FUNCTION_BLOCK xPlanarControl
VAR
	
	_PlanarMover			: ARRAY [1..MoverCount] OF MC_PlanarMover;
	_PlanarFeedback			: ARRAY [1..MoverCount] OF MC_PlanarFeedback;
	_MoveParameters			: ARRAY [1..MoverCount] OF ST_MoverParameters;
	
	_i						: BYTE;
	_LocalState				: BYTE;
	_InternalCounter		: UINT;
	_ErrorCount				: UINT;
	_CommandDone			: BOOL;
	
	_Enabled				: ARRAY [1.._MoverCount] OF BOOL;
	_Error					: ARRAY [1.._MoverCount] OF BOOL;
	_Busy					: ARRAY [1.._MoverCount] OF BOOL;
	_Done					: ARRAY [1.._MoverCount] OF BOOL;
	
	_Velocity				: LREAL := 2000;
	_Acceleration			: LREAL := 20000;
	_Deceleration			: LREAL := 20000;
	_Jerk					: LREAL := 200000;
	_NumberOfRotations		: UDINT := 5;
	
END_VAR
VAR CONSTANT
	
	_MoverCount				: BYTE := 2;

END_VAR

// NETWORK 1

METHOD CyclicUpdate : BOOL
VAR_INPUT
END_VAR

FOR _i := 1 TO _MoverCount DO
	
	_PlanarMover[_i].Update();
	_PlanarFeedback[_i].Update();
	
	IF _PlanarMover[_i].MCTOPLC.STD.State = 3 THEN
		_Enabled[_i] := TRUE;
	ELSE
		_Enabled[_i] := FALSE;
	END_IF

	_Error[_i] := _PlanarFeedback[_i].Error;
	_Busy[_i] := _PlanarFeedback[_i].Busy;
	_Done[_i] := _PlanarFeedback[_i].Done;
	
END_FOR

_MoveParameters[1].Options.useOrientation := TRUE;
_MoveParameters[1].Constraints.SetValuesVADJ(V := _Velocity, A := _Acceleration, D := _Deceleration, J := _Jerk);
_MoveParameters[1].rotateOptions.additionalTurns := _NumberOfRotations;
_MoveParameters[1].rotateOptions.direction := 1;

_MoveParameters[2].Options.useOrientation := TRUE;
_MoveParameters[2].Constraints.SetValuesVADJ(V := _Velocity, A := _Acceleration, D := _Deceleration, J := _Jerk);
_MoveParameters[2].rotateOptions.additionalTurns := _NumberOfRotations;
_MoveParameters[2].rotateOptions.direction := 3;
END_METHOD

METHOD PUBLIC DecreaseMoverHeight : BOOL
VAR_INPUT
END_VAR

// Movers go a bit low
	
CASE _LocalState OF
	
	0:
		_LocalState := 1;
	
	1:
		FOR _i := 1 TO _MoverCount DO
			_PlanarMover[_i].MoveZ
			(	
				commandFeedback		:= _PlanarFeedback[_i],
				targetPosition		:= 2.0,
				constraint			:= _MoveParameters[_i].Constraints
			);
		END_FOR
		_LocalState := 2;
	
	2:
		_CommandDone := TRUE;
		FOR _i := 1 TO _MoverCount DO
			IF NOT(_PlanarFeedback[_i].Done) THEN
				_CommandDone := FALSE;
				_InternalCounter := _InternalCounter + 1;
			END_IF
		END_FOR
		
		IF _InternalCounter >= 10000 THEN
			_LocalState := 0;
			_InternalCounter := 0;
			DecreaseMoverHeight := FALSE;
		END_IF
		
		IF _CommandDone THEN
			_CommandDone := FALSE;
			_InternalCounter := 0;
			_LocalState := 2;
		END_IF

	3:
		DecreaseMoverHeight := TRUE;
		_LocalState := 0;

END_CASE
END_METHOD

METHOD DetectErrors : BOOL
VAR_INPUT
END_VAR

FOR _i := 1 TO _MoverCount DO
	IF _PlanarMover[_i].Error THEN
		_Error[_i] := TRUE;
		_ErrorCount := _ErrorCount + 1;
		DetectErrors := TRUE;
	END_IF
END_FOR
END_METHOD

METHOD DisableMovers : BOOL
VAR_INPUT
END_VAR

CASE _LocalState OF
	
	0:
		FOR _i := 1 TO _MoverCount DO
			_PlanarMover[_i].Disable(_PlanarFeedback[_i]);
		END_FOR
		_LocalState := 1;
	
	1:
		_CommandDone := TRUE;
		FOR _i := 1 TO _MoverCount DO
			IF NOT(_PlanarFeedback[_i].Done) THEN
				_CommandDone := FALSE;
				_InternalCounter := _InternalCounter + 1;
			END_IF
		END_FOR
		
		IF _InternalCounter >= 10000 THEN
			_LocalState := 0;
			_InternalCounter := 0;
			DisableMovers := FALSE;
		END_IF
		
		IF _CommandDone THEN
			_CommandDone := FALSE;
			_InternalCounter := 0;
			_LocalState := 2;
		END_IF
	
	2:
		_LocalState := 0;
		DisableMovers := TRUE;

END_CASE
END_METHOD

METHOD EnableMovers : BOOL
VAR_INPUT
END_VAR

CASE _LocalState OF
	
	0:
		FOR _i := 1 TO _MoverCount DO
			_PlanarMover[_i].Enable(_PlanarFeedback[_i]);
		END_FOR
		_LocalState := 1;
	
	1:
		_CommandDone := TRUE;
		FOR _i := 1 TO _MoverCount DO
			IF NOT(_PlanarFeedback[_i].Done) THEN
				_CommandDone := FALSE;
				_InternalCounter := _InternalCounter + 1;
			END_IF
		END_FOR
		
		IF _InternalCounter >= 10000 THEN
			_LocalState := 0;
			_InternalCounter := 0;
			EnableMovers := FALSE;
		END_IF
		
		IF _CommandDone THEN
			_CommandDone := FALSE;
			_InternalCounter := 0;
			_LocalState := 2;
		END_IF
	
	2:
		_LocalState := 0;
		EnableMovers := TRUE;

END_CASE
END_METHOD

METHOD PUBLIC FollowTileEdge : BOOL
VAR_INPUT
END_VAR

// Movers move to edge of tiles and follow the perimeter, then move to home
	
	CASE _LocalState OF
		
		0:
			_LocalState := 1;
	
		1:
			_MoveParameters[1].targetPosition.x := 180;
			_MoveParameters[1].targetPosition.y := 183;
			_MoveParameters[2].targetPosition.x := 296;
			_MoveParameters[2].targetPosition.y := 183;
			_LocalState := 2;
		
		2:
			FOR _i := 1 TO _MoverCount DO
				_PlanarMover[_i].MoveToPosition
				(
					commandFeedback 	:= _PlanarFeedback[_i],
					targetPosition 		:= _MoveParameters[_i].targetPosition,
					constraint 			:= _MoveParameters[_i].Constraints,
					options 			:= _MoveParameters[_i].Options
				);
			END_FOR
			_LocalState := 3;
		
		3:
			_CommandDone := TRUE;
			FOR _i := 1 TO _MoverCount DO
				IF NOT(_PlanarFeedback[_i].Done) THEN
					_CommandDone := FALSE;
					_InternalCounter := _InternalCounter + 1;
				END_IF
			END_FOR
			
			IF _InternalCounter >= 10000 THEN
				_LocalState := 0;
				_InternalCounter := 0;
				FollowTileEdge := FALSE;
			END_IF
			
			IF _CommandDone THEN
				_CommandDone := FALSE;
				_InternalCounter := 0;
				_LocalState := 4;
			END_IF
	
		4:
			_MoveParameters[1].targetPosition.x := 57;
			_MoveParameters[1].targetPosition.y := 183;
			_MoveParameters[2].targetPosition.x := 423;
			_MoveParameters[2].targetPosition.y := 183;
			_LocalState := 5;
		
		5:
			FOR _i := 1 TO _MoverCount DO
				_PlanarMover[_i].MoveToPosition
				(
					commandFeedback 	:= _PlanarFeedback[_i],
					targetPosition 		:= _MoveParameters[_i].targetPosition,
					constraint 			:= _MoveParameters[_i].Constraints,
					options 			:= _MoveParameters[_i].Options
				);
			END_FOR
			_LocalState := 6;
		
		6:
			_CommandDone := TRUE;
			FOR _i := 1 TO _MoverCount DO
				IF NOT(_PlanarFeedback[_i].Done) THEN
					_CommandDone := FALSE;
					_InternalCounter := _InternalCounter + 1;
				END_IF
			END_FOR
			
			IF _InternalCounter >= 10000 THEN
				_LocalState := 0;
				_InternalCounter := 0;
				FollowTileEdge := FALSE;
			END_IF
			
			IF _CommandDone THEN
				_CommandDone := FALSE;
				_InternalCounter := 0;
				_LocalState := 7;
			END_IF
			
		7:
			_MoveParameters[1].targetPosition.x := 57;
			_MoveParameters[1].targetPosition.y := 57;
			_MoveParameters[2].targetPosition.x := 423;
			_MoveParameters[2].targetPosition.y := 57;
			_LocalState := 8;
		
		8:
			FOR _i := 1 TO _MoverCount DO
				_PlanarMover[_i].MoveToPosition
				(
					commandFeedback 	:= _PlanarFeedback[_i],
					targetPosition 		:= _MoveParameters[_i].targetPosition,
					constraint 			:= _MoveParameters[_i].Constraints,
					options 			:= _MoveParameters[_i].Options
				);
			END_FOR
			_LocalState := 9;
		
		9:
			_CommandDone := TRUE;
			FOR _i := 1 TO _MoverCount DO
				IF NOT(_PlanarFeedback[_i].Done) THEN
					_CommandDone := FALSE;
					_InternalCounter := _InternalCounter + 1;
				END_IF
			END_FOR
			
			IF _InternalCounter >= 10000 THEN
				_LocalState := 0;
				_InternalCounter := 0;
				FollowTileEdge := FALSE;
			END_IF
			
			IF _CommandDone THEN
				_CommandDone := FALSE;
				_InternalCounter := 0;
				_LocalState := 10;
			END_IF
			
		10:
			_MoveParameters[1].targetPosition.x := 180;
			_MoveParameters[1].targetPosition.y := 57;
			_MoveParameters[2].targetPosition.x := 296;
			_MoveParameters[2].targetPosition.y := 57;
			_LocalState := 11;
		
		11:
			FOR _i := 1 TO _MoverCount DO
				_PlanarMover[_i].MoveToPosition
				(
					commandFeedback 	:= _PlanarFeedback[_i],
					targetPosition 		:= _MoveParameters[_i].targetPosition,
					constraint 			:= _MoveParameters[_i].Constraints,
					options 			:= _MoveParameters[_i].Options
				);
			END_FOR
			_LocalState := 12;
		
		12:
			_CommandDone := TRUE;
			FOR _i := 1 TO _MoverCount DO
				IF NOT(_PlanarFeedback[_i].Done) THEN
					_CommandDone := FALSE;
					_InternalCounter := _InternalCounter + 1;
				END_IF
			END_FOR
			
			IF _InternalCounter >= 10000 THEN
				_LocalState := 0;
				_InternalCounter := 0;
				FollowTileEdge := FALSE;
			END_IF
			
			IF _CommandDone THEN
				_CommandDone := FALSE;
				_InternalCounter := 0;
				_LocalState := 13;
			END_IF
			
		13:
			_MoveParameters[1].targetPosition.x := 120;
			_MoveParameters[1].targetPosition.y := 120;
			_MoveParameters[2].targetPosition.x := 360;
			_MoveParameters[2].targetPosition.y := 120;
			_LocalState := 14;
		
		14:
			FOR _i := 1 TO _MoverCount DO
				_PlanarMover[_i].MoveToPosition
				(
					commandFeedback 	:= _PlanarFeedback[_i],
					targetPosition 		:= _MoveParameters[_i].targetPosition,
					constraint 			:= _MoveParameters[_i].Constraints,
					options 			:= _MoveParameters[_i].Options
				);
			END_FOR
			_LocalState := 15;
		
		15:
			_CommandDone := TRUE;
			FOR _i := 1 TO _MoverCount DO
				IF NOT(_PlanarFeedback[_i].Done) THEN
					_CommandDone := FALSE;
					_InternalCounter := _InternalCounter + 1;
				END_IF
			END_FOR
			
			IF _InternalCounter >= 10000 THEN
				_LocalState := 0;
				_InternalCounter := 0;
				FollowTileEdge := FALSE;
			END_IF
			
			IF _CommandDone THEN
				_CommandDone := FALSE;
				_InternalCounter := 0;
				_LocalState := 16;
			END_IF
			
		16:
			FollowTileEdge := TRUE;
			_LocalState := 0;
			
	END_CASE
END_METHOD

METHOD PUBLIC Home : BOOL
VAR_INPUT
END_VAR

// Move movers to the middle of tiles.
	
CASE _LocalState OF
		
	0:
		_LocalState := 1;
		
	1:
		_MoveParameters[1].targetPosition.x := 120;
		_MoveParameters[1].targetPosition.y := 120;
		_MoveParameters[2].targetPosition.x := 360;
		_MoveParameters[2].targetPosition.y := 120;
		_LocalState := 2;
		
	2:
		FOR _i := 1 TO _MoverCount DO
			_PlanarMover[_i].MoveToPosition
			(
				commandFeedback 	:= _PlanarFeedback[_i],
				targetPosition 		:= _MoveParameters[_i].targetPosition,
				constraint 			:= _MoveParameters[_i].Constraints,
				options 			:= _MoveParameters[_i].Options
			);
		END_FOR
		_LocalState := 3;
		
	3:
		_CommandDone := TRUE;
		FOR _i := 1 TO _MoverCount DO
			IF NOT(_PlanarFeedback[_i].Done) THEN
				_CommandDone := FALSE;
				_InternalCounter := _InternalCounter + 1;
			END_IF
		END_FOR
		
		IF _InternalCounter >= 10000 THEN
			_LocalState := 0;
			_InternalCounter := 0;
			Home := FALSE;
		END_IF
		
		IF _CommandDone THEN
			_CommandDone := FALSE;
			_InternalCounter := 0;
			_LocalState := 4;
		END_IF
		
	4:
		Home := TRUE;
		_LocalState := 0;
		
		
END_CASE
END_METHOD

PROPERTY MoverAcceleration : LREAL
GET
MoverAcceleration := _Acceleration;
END_GET
SET
IF (MoverAcceleration <= 0) OR (MoverAcceleration > 20000) THEN
	_Acceleration := 20000;
ELSE
	_Acceleration := MoverAcceleration;
END_IF
END_SET
END_PROPERTY

PROPERTY MoverDeceleration : LREAL
GET
MoverDeceleration := _Deceleration;
END_GET
SET
IF (MoverDeceleration <= 0) OR (MoverDeceleration > 20000) THEN
	_Deceleration := 20000;
ELSE
	_Deceleration := MoverDeceleration;
END_IF
END_SET
END_PROPERTY

PROPERTY MoverJerk : LREAL
GET
MoverJerk := _Jerk;
END_GET
SET
IF (MoverJerk <= 0) OR (MoverJerk > 200000) THEN
	_Jerk := 200000;
ELSE
	_Jerk := MoverJerk;
END_IF
END_SET
END_PROPERTY

PROPERTY MoverVelocity : LREAL
GET
MoverVelocity := _Velocity;
END_GET
SET
IF (MoverVelocity <= 0) OR (MoverVelocity > 2000) THEN
	_Velocity := 2000;
ELSE
	_Velocity := MoverVelocity;
END_IF
END_SET
END_PROPERTY

PROPERTY NumberOfRotations : UDINT
GET
NumberOfRotations := _NumberOfRotations;
END_GET
SET
IF (NumberOfRotations <= 0) THEN
	_NumberOfRotations := 1;
ELSE
	_NumberOfRotations := NumberOfRotations;
END_IF
END_SET
END_PROPERTY

METHOD ResetErrors : BOOL
VAR_INPUT
END_VAR

CASE _LocalState OF
	
	0: 
		FOR _i := 1 TO _MoverCount DO
			_PlanarMover[_i].Reset(_PlanarFeedback[_i]);
		END_FOR
		_LocalState := 1;
	
	1:	
		_CommandDone := TRUE;
		FOR _i := 1 TO _MoverCount DO
			IF NOT(_PlanarFeedback[_i].Done) THEN
				_CommandDone := FALSE;
				_InternalCounter := _InternalCounter + 1;
			END_IF
		END_FOR
		
		IF _InternalCounter >= 10000 THEN
			_LocalState := 0;
			_InternalCounter := 0;
			ResetErrors := FALSE;
		END_IF
		
		IF _CommandDone THEN
			_CommandDone := FALSE;
			_InternalCounter := 0;
			_LocalState := 2;
		END_IF

			
	2:
		_LocalState := 0;
		ResetErrors := TRUE;
	
END_CASE
END_METHOD

METHOD PUBLIC Spin : BOOL
VAR_INPUT
END_VAR

// Movers spin

CASE _LocalState OF
	
	0:
		_LocalState := 1;

	
	1:
		FOR _i := 1 TO _MoverCount DO
			_PlanarMover[_i].MoveC
			(	
				commandFeedback		:= _PlanarFeedback[_i],
				targetPosition		:= 0,
				constraint			:= _MoveParameters[_i].Constraints,
				options 			:= _MoveParameters[_i].rotateOptions
			);
		END_FOR
		_LocalState := 2;
	
	2:
		_CommandDone := TRUE;
		FOR _i := 1 TO _MoverCount DO
			IF NOT(_PlanarFeedback[_i].Done) THEN
				_CommandDone := FALSE;
				_InternalCounter := _InternalCounter + 1;
			END_IF
		END_FOR
		
		IF _InternalCounter >= 10000 THEN
			_LocalState := 0;
			_InternalCounter := 0;
			Spin := FALSE;
		END_IF
		
		IF _CommandDone THEN
			_CommandDone := FALSE;
			_InternalCounter := 0;
			_LocalState := 2;
		END_IF
		
	3:
		Spin := TRUE;
		_LocalState := 0;
	
END_CASE
END_METHOD

METHOD PUBLIC SwapPlaces : BOOL
VAR_INPUT
END_VAR

// Movers swap tiles, then swap back, then move to home
	
CASE _LocalState OF
	
	0:
		_LocalState := 1;

	1:
		_MoveParameters[1].targetPosition.x := 175;
		_MoveParameters[1].targetPosition.y := 183;
		_MoveParameters[2].targetPosition.x := 301;
		_MoveParameters[2].targetPosition.y := 57;
		_LocalState := 2;
	
	2:
		FOR _i := 1 TO _MoverCount DO
			_PlanarMover[_i].MoveToPosition
			(
				commandFeedback 	:= _PlanarFeedback[_i],
				targetPosition 		:= _MoveParameters[_i].targetPosition,
				constraint 			:= _MoveParameters[_i].Constraints,
				options 			:= _MoveParameters[_i].Options
			);
		END_FOR
		_LocalState := 3;
	
	3:
		_CommandDone := TRUE;
		FOR _i := 1 TO _MoverCount DO
			IF NOT(_PlanarFeedback[_i].Done) THEN
				_CommandDone := FALSE;
				_InternalCounter := _InternalCounter + 1;
			END_IF
		END_FOR
		
		IF _InternalCounter >= 10000 THEN
			_LocalState := 0;
			_InternalCounter := 0;
			SwapPlaces := FALSE;
		END_IF
		
		IF _CommandDone THEN
			_CommandDone := FALSE;
			_InternalCounter := 0;
			_LocalState := 4;
		END_IF

	4:
		_MoveParameters[1].targetPosition.x := 301;
		_MoveParameters[1].targetPosition.y := 183;
		_MoveParameters[2].targetPosition.x := 175;
		_MoveParameters[2].targetPosition.y := 57;
		_LocalState := 5;
	
	5:
		FOR _i := 1 TO _MoverCount DO
			_PlanarMover[_i].MoveToPosition
			(
				commandFeedback 	:= _PlanarFeedback[_i],
				targetPosition 		:= _MoveParameters[_i].targetPosition,
				constraint 			:= _MoveParameters[_i].Constraints,
				options 			:= _MoveParameters[_i].Options
			);
		END_FOR
		_LocalState := 6;
	
	6:
		_CommandDone := TRUE;
		FOR _i := 1 TO _MoverCount DO
			IF NOT(_PlanarFeedback[_i].Done) THEN
				_CommandDone := FALSE;
				_InternalCounter := _InternalCounter + 1;
			END_IF
		END_FOR
		
		IF _InternalCounter >= 10000 THEN
			_LocalState := 0;
			_InternalCounter := 0;
			SwapPlaces := FALSE;
		END_IF
		
		IF _CommandDone THEN
			_CommandDone := FALSE;
			_InternalCounter := 0;
			_LocalState := 7;
		END_IF
		
	7:
		_MoveParameters[1].targetPosition.x := 301;
		_MoveParameters[1].targetPosition.y := 57;
		_MoveParameters[2].targetPosition.x := 175;
		_MoveParameters[2].targetPosition.y := 183;
		_LocalState := 8;
	
	8:
		FOR _i := 1 TO _MoverCount DO
			_PlanarMover[_i].MoveToPosition
			(
				commandFeedback 	:= _PlanarFeedback[_i],
				targetPosition 		:= _MoveParameters[_i].targetPosition,
				constraint 			:= _MoveParameters[_i].Constraints,
				options 			:= _MoveParameters[_i].Options
			);
		END_FOR
		_LocalState := 9;
	
	9:
		_CommandDone := TRUE;
		FOR _i := 1 TO _MoverCount DO
			IF NOT(_PlanarFeedback[_i].Done) THEN
				_CommandDone := FALSE;
				_InternalCounter := _InternalCounter + 1;
			END_IF
		END_FOR
		
		IF _InternalCounter >= 10000 THEN
			_LocalState := 0;
			_InternalCounter := 0;
			SwapPlaces := FALSE;
		END_IF
		
		IF _CommandDone THEN
			_CommandDone := FALSE;
			_InternalCounter := 0;
			_LocalState := 10;
		END_IF
		
	10:
		_MoveParameters[1].targetPosition.x := 175;
		_MoveParameters[1].targetPosition.y := 57;
		_MoveParameters[2].targetPosition.x := 301;
		_MoveParameters[2].targetPosition.y := 183;
		_LocalState := 11;
	
	11:
		FOR _i := 1 TO _MoverCount DO
			_PlanarMover[_i].MoveToPosition
			(
				commandFeedback 	:= _PlanarFeedback[_i],
				targetPosition 		:= _MoveParameters[_i].targetPosition,
				constraint 			:= _MoveParameters[_i].Constraints,
				options 			:= _MoveParameters[_i].Options
			);
		END_FOR
		_LocalState := 12;
	
	12:
		_CommandDone := TRUE;
		FOR _i := 1 TO _MoverCount DO
			IF NOT(_PlanarFeedback[_i].Done) THEN
				_CommandDone := FALSE;
				_InternalCounter := _InternalCounter + 1;
			END_IF
		END_FOR
		
		IF _InternalCounter >= 10000 THEN
			_LocalState := 0;
			_InternalCounter := 0;
			SwapPlaces := FALSE;
		END_IF
		
		IF _CommandDone THEN
			_CommandDone := FALSE;
			_InternalCounter := 0;
			_LocalState := 13;
		END_IF
		
	13:
		_MoveParameters[1].targetPosition.x := 120;
		_MoveParameters[1].targetPosition.y := 120;
		_MoveParameters[2].targetPosition.x := 360;
		_MoveParameters[2].targetPosition.y := 120;
		_LocalState := 14;
	
	14:
		FOR _i := 1 TO _MoverCount DO
			_PlanarMover[_i].MoveToPosition
			(
				commandFeedback 	:= _PlanarFeedback[_i],
				targetPosition 		:= _MoveParameters[_i].targetPosition,
				constraint 			:= _MoveParameters[_i].Constraints,
				options 			:= _MoveParameters[_i].Options
			);
		END_FOR
		_LocalState := 15;
	
	15:
		_CommandDone := TRUE;
		FOR _i := 1 TO _MoverCount DO
			IF NOT(_PlanarFeedback[_i].Done) THEN
				_CommandDone := FALSE;
				_InternalCounter := _InternalCounter + 1;
			END_IF
		END_FOR
		
		IF _InternalCounter >= 10000 THEN
			_LocalState := 0;
			_InternalCounter := 0;
			SwapPlaces := FALSE;
		END_IF
		
		IF _CommandDone THEN
			_CommandDone := FALSE;
			_InternalCounter := 0;
			_LocalState := 16;
		END_IF
		
	16:
		SwapPlaces := TRUE;
		_LocalState := 0;
		
END_CASE
END_METHOD

METHOD PUBLIC Tilt : BOOL
VAR_INPUT
END_VAR

// Movers tilt

CASE _LocalState OF
	
	0:
		_LocalState := 1;
		
	1:
		FOR _i := 1 TO _MoverCount DO
			_PlanarMover[_i].MoveZ
			(	
				commandFeedback		:= _PlanarFeedback[_i],
				targetPosition		:= 5.0,
				constraint			:= _MoveParameters[_i].Constraints
			);
		END_FOR
		_LocalState := 2;
	
	2:
		_CommandDone := TRUE;
		FOR _i := 1 TO _MoverCount DO
			IF NOT(_PlanarFeedback[_i].Done) THEN
				_CommandDone := FALSE;
				_InternalCounter := _InternalCounter + 1;
			END_IF
		END_FOR
		
		IF _InternalCounter >= 10000 THEN
			_LocalState := 0;
			_InternalCounter := 0;
			Tilt := FALSE;
		END_IF
		
		IF _CommandDone THEN
			_CommandDone := FALSE;
			_InternalCounter := 0;
			_LocalState := 3;
		END_IF

	
	3:
		FOR _i := 1 TO xPlanarLink.MoverCount DO
			xPlanarLink.PlanarMover[_i].MoveA
			(	
				commandFeedback		:= xPlanarLink.PlanarFeedback[_i],
				targetPosition		:= 4.0,
				constraint			:= _MoveParameters[_i].Constraints
			);
		END_FOR
		_LocalState := 4;
	
	4:
		_CommandDone := TRUE;
		FOR _i := 1 TO _MoverCount DO
			IF NOT(_PlanarFeedback[_i].Done) THEN
				_CommandDone := FALSE;
				_InternalCounter := _InternalCounter + 1;
			END_IF
		END_FOR
		
		IF _InternalCounter >= 10000 THEN
			_LocalState := 0;
			_InternalCounter := 0;
			Tilt := FALSE;
		END_IF
		
		IF _CommandDone THEN
			_CommandDone := FALSE;
			_InternalCounter := 0;
			_LocalState := 5;
		END_IF
		
	5:
		FOR _i := 1 TO _MoverCount DO
			_PlanarMover[_i].MoveA
			(	
				commandFeedback		:= _PlanarFeedback[_i],
				targetPosition		:= -4.0,
				constraint			:= _MoveParameters[_i].Constraints
			);
		END_FOR
		_LocalState := 6;
	
	6:
		_CommandDone := TRUE;
		FOR _i := 1 TO _MoverCount DO
			IF NOT(_PlanarFeedback[_i].Done) THEN
				_CommandDone := FALSE;
				_InternalCounter := _InternalCounter + 1;
			END_IF
		END_FOR
		
		IF _InternalCounter >= 10000 THEN
			_LocalState := 0;
			_InternalCounter := 0;
			Tilt := FALSE;
		END_IF
		
		IF _CommandDone THEN
			_CommandDone := FALSE;
			_InternalCounter := 0;
			_LocalState := 7;
		END_IF
	
	7:
		FOR _i := 1 TO _MoverCount DO
			_PlanarMover[_i].MoveA
			(	
				commandFeedback		:= _PlanarFeedback[_i],
				targetPosition		:= 0.0,
				constraint			:= _MoveParameters[_i].Constraints
			);
		END_FOR
		_LocalState := 8;
	
	8:
		_CommandDone := TRUE;
		FOR _i := 1 TO _MoverCount DO
			IF NOT(_PlanarFeedback[_i].Done) THEN
				_CommandDone := FALSE;
				_InternalCounter := _InternalCounter + 1;
			END_IF
		END_FOR
		
		IF _InternalCounter >= 10000 THEN
			_LocalState := 0;
			_InternalCounter := 0;
			Tilt := FALSE;
		END_IF
		
		IF _CommandDone THEN
			_CommandDone := FALSE;
			_InternalCounter := 0;
			_LocalState := 9;
		END_IF
		
	9:
		FOR _i := 1 TO _MoverCount DO
			_PlanarMover[_i].MoveB
			(	
				commandFeedback		:= _PlanarFeedback[_i],
				targetPosition		:= 4.0,
				constraint			:= _MoveParameters[_i].Constraints
			);
		END_FOR
		_LocalState := 10;
	
	10:
		_CommandDone := TRUE;
		FOR _i := 1 TO _MoverCount DO
			IF NOT(_PlanarFeedback[_i].Done) THEN
				_CommandDone := FALSE;
				_InternalCounter := _InternalCounter + 1;
			END_IF
		END_FOR
		
		IF _InternalCounter >= 10000 THEN
			_LocalState := 0;
			_InternalCounter := 0;
			Tilt := FALSE;
		END_IF
		
		IF _CommandDone THEN
			_CommandDone := FALSE;
			_InternalCounter := 0;
			_LocalState := 11;
		END_IF
		
	11:
		FOR _i := 1 TO _MoverCount DO
			_PlanarMover[_i].MoveB
			(	
				commandFeedback		:= _PlanarFeedback[_i],
				targetPosition		:= -4.0,
				constraint			:= _MoveParameters[_i].Constraints
			);
		END_FOR
		_LocalState := 12;
	
	12:
		_CommandDone := TRUE;
		FOR _i := 1 TO _MoverCount DO
			IF NOT(_PlanarFeedback[_i].Done) THEN
				_CommandDone := FALSE;
				_InternalCounter := _InternalCounter + 1;
			END_IF
		END_FOR
		
		IF _InternalCounter >= 10000 THEN
			_LocalState := 0;
			_InternalCounter := 0;
			Tilt := FALSE;
		END_IF
		
		IF _CommandDone THEN
			_CommandDone := FALSE;
			_InternalCounter := 0;
			_LocalState := 13;
		END_IF
	
	13:
		FOR _i := 1 TO _MoverCount DO
			_PlanarMover[_i].MoveB
			(	
				commandFeedback		:= _PlanarFeedback[_i],
				targetPosition		:= 0.0,
				constraint			:= _MoveParameters[_i].Constraints
			);
		END_FOR
		_LocalState := 14;
	
	14:
		_CommandDone := TRUE;
		FOR _i := 1 TO _MoverCount DO
			IF NOT(_PlanarFeedback[_i].Done) THEN
				_CommandDone := FALSE;
				_InternalCounter := _InternalCounter + 1;
			END_IF
		END_FOR
		
		IF _InternalCounter >= 10000 THEN
			_LocalState := 0;
			_InternalCounter := 0;
			Tilt := FALSE;
		END_IF
		
		IF _CommandDone THEN
			_CommandDone := FALSE;
			_InternalCounter := 0;
			_LocalState := 15;
		END_IF
		
	15:
		FOR _i := 1 TO _MoverCount DO
			_PlanarMover[_i].MoveZ
			(	
				commandFeedback		:= _PlanarFeedback[_i],
				targetPosition		:= 2.0,
				constraint			:= _MoveParameters[_i].Constraints
			);
		END_FOR
		_LocalState := 16;
	
	16:
		_CommandDone := TRUE;
		FOR _i := 1 TO _MoverCount DO
			IF NOT(_PlanarFeedback[_i].Done) THEN
				_CommandDone := FALSE;
				_InternalCounter := _InternalCounter + 1;
			END_IF
		END_FOR
		
		IF _InternalCounter >= 10000 THEN
			_LocalState := 0;
			_InternalCounter := 0;
			Tilt := FALSE;
		END_IF
		
		IF _CommandDone THEN
			_CommandDone := FALSE;
			_InternalCounter := 0;
			_LocalState := 17;
		END_IF
		
	17:
		Tilt := TRUE;
		_LocalState := 0;
	
END_CASE
END_METHOD

METHOD PUBLIC VaryMoverHeight : BOOL
VAR_INPUT
END_VAR

// Movers go a bit high

CASE _LocalState OF
	
	0:
		_LocalState := 1;
	
	1:
		FOR _i := 1 TO _MoverCount DO
			_PlanarMover[_i].MoveZ
			(	
				commandFeedback		:= _PlanarFeedback[_i],
				targetPosition		:= 5.0,
				constraint			:= _MoveParameters[_i].Constraints
			);
		END_FOR
		_LocalState := 2;
	
	2:
		_CommandDone := TRUE;
		FOR _i := 1 TO _MoverCount DO
			IF NOT(_PlanarFeedback[_i].Done) THEN
				_CommandDone := FALSE;
				_InternalCounter := _InternalCounter + 1;
			END_IF
		END_FOR
		
		IF _InternalCounter >= 10000 THEN
			_LocalState := 0;
			_InternalCounter := 0;
			VaryMoverHeight := FALSE;
		END_IF
		
		IF _CommandDone THEN
			_CommandDone := FALSE;
			_InternalCounter := 0;
			_LocalState := 3;
		END_IF
		
	3:
		FOR _i := 1 TO _MoverCount DO
			_PlanarMover[_i].MoveZ
			(	
				commandFeedback		:= _PlanarFeedback[_i],
				targetPosition		:= 2.0,
				constraint			:= _MoveParameters[_i].Constraints
			);
		END_FOR
		_LocalState := 4;
	
	4:
		_CommandDone := TRUE;
		FOR _i := 1 TO _MoverCount DO
			IF NOT(_PlanarFeedback[_i].Done) THEN
				_CommandDone := FALSE;
				_InternalCounter := _InternalCounter + 1;
			END_IF
		END_FOR
		
		IF _InternalCounter >= 10000 THEN
			_LocalState := 0;
			_InternalCounter := 0;
			VaryMoverHeight := FALSE;
		END_IF
		
		IF _CommandDone THEN
			_CommandDone := FALSE;
			_InternalCounter := 0;
			_LocalState := 5;
		END_IF
		
	5:
		FOR _i := 1 TO _MoverCount DO
			_PlanarMover[_i].MoveZ
			(	
				commandFeedback		:= _PlanarFeedback[_i],
				targetPosition		:= 5.0,
				constraint			:= _MoveParameters[_i].Constraints
			);
		END_FOR
		_LocalState := 6;
	
	6:
		_CommandDone := TRUE;
		FOR _i := 1 TO _MoverCount DO
			IF NOT(_PlanarFeedback[_i].Done) THEN
				_CommandDone := FALSE;
				_InternalCounter := _InternalCounter + 1;
			END_IF
		END_FOR
		
		IF _InternalCounter >= 10000 THEN
			_LocalState := 0;
			_InternalCounter := 0;
			VaryMoverHeight := FALSE;
		END_IF
		
		IF _CommandDone THEN
			_CommandDone := FALSE;
			_InternalCounter := 0;
			_LocalState := 7;
		END_IF
		
	7:
		FOR _i := 1 TO _MoverCount DO
			_PlanarMover[_i].MoveZ
			(	
				commandFeedback		:= _PlanarFeedback[_i],
				targetPosition		:= 2.0,
				constraint			:= _MoveParameters[_i].Constraints
			);
		END_FOR
		_LocalState := 8;
	
	8:
		_CommandDone := TRUE;
		FOR _i := 1 TO _MoverCount DO
			IF NOT(_PlanarFeedback[_i].Done) THEN
				_CommandDone := FALSE;
				_InternalCounter := _InternalCounter + 1;
			END_IF
		END_FOR
		
		IF _InternalCounter >= 10000 THEN
			_LocalState := 0;
			_InternalCounter := 0;
			VaryMoverHeight := FALSE;
		END_IF
		
		IF _CommandDone THEN
			_CommandDone := FALSE;
			_InternalCounter := 0;
			_LocalState := 9;
		END_IF
		
	9:
		FOR _i := 1 TO _MoverCount DO
			_PlanarMover[_i].MoveZ
			(	
				commandFeedback		:= _PlanarFeedback[_i],
				targetPosition		:= 5.0,
				constraint			:= _MoveParameters[_i].Constraints
			);
		END_FOR
		_LocalState := 10;
	
	10:
		_CommandDone := TRUE;
		FOR _i := 1 TO _MoverCount DO
			IF NOT(_PlanarFeedback[_i].Done) THEN
				_CommandDone := FALSE;
				_InternalCounter := _InternalCounter + 1;
			END_IF
		END_FOR
		
		IF _InternalCounter >= 10000 THEN
			_LocalState := 0;
			_InternalCounter := 0;
			VaryMoverHeight := FALSE;
		END_IF
		
		IF _CommandDone THEN
			_CommandDone := FALSE;
			_InternalCounter := 0;
			_LocalState := 11;
		END_IF

	11:
		FOR _i := 1 TO _MoverCount DO
			_PlanarMover[_i].MoveZ
			(	
				commandFeedback		:= _PlanarFeedback[_i],
				targetPosition		:= 2.0,
				constraint			:= _MoveParameters[_i].Constraints
			);
		END_FOR
		_LocalState := 12;
	
	12:
		_CommandDone := TRUE;
		FOR _i := 1 TO _MoverCount DO
			IF NOT(_PlanarFeedback[_i].Done) THEN
				_CommandDone := FALSE;
				_InternalCounter := _InternalCounter + 1;
			END_IF
		END_FOR
		
		IF _InternalCounter >= 10000 THEN
			_LocalState := 0;
			_InternalCounter := 0;
			VaryMoverHeight := FALSE;
		END_IF
		
		IF _CommandDone THEN
			_CommandDone := FALSE;
			_InternalCounter := 0;
			_LocalState := 13;
		END_IF
		
	13:
		VaryMoverHeight := TRUE;
		_LocalState := 0;

END_CASE
END_METHOD

END_FUNCTION_BLOCK

(* stored: Version 1.1.0.1, ProductVersion 3.1.4024.12
   POU xPlanarControl: Id {418f5a4e-4a80-43af-8346-cac2175cf5a1}, SpecialFunc None
   Folder Movements 2-Tile: Id {564f56f8-bb5c-4eca-8a56-c64a7594c15d}
   Folder Movements General: Id {aee95a18-140d-4ee9-ac40-69e7d69f9acf}
   Folder Power and Utility: Id {c5ba77ca-a5ce-43bc-a81f-9b9628e1d54c}
   Folder Properties: Id {0453768e-2223-4ce2-b57c-26f2fb086bed}
   Method CyclicUpdate: Id {c7e9e683-b8ab-4217-b047-2e15baa6471c}
   Method DecreaseMoverHeight: Id {d9c1f541-a92b-457b-b498-ae0f9078990c}
   Method DetectErrors: Id {daaeb43c-d127-4004-8d5e-5bf5a68f458b}
   Method DisableMovers: Id {425fd2bc-6f54-4fce-935d-1f0a1dc8c22b}
   Method EnableMovers: Id {ecc31ae1-6e60-4543-ab06-14adb5849eca}
   Method FollowTileEdge: Id {87cfbbfe-b39c-4b51-8245-78953324c448}
   Method Home: Id {c3147f7b-df53-4a91-a0c1-7a36cd9f6a0f}
   Property MoverAcceleration: Id {46b26c09-adf7-42f2-a584-23d59417babe}
   Get Get: Id {f150d898-6fb7-4350-b36b-5cbdc8b0e614}
   Set Set: Id {1e98ee18-12de-4aa7-9a0d-740e3225678d}
   Property MoverDeceleration: Id {6dc3dcb8-27e4-496b-9d9d-8aa4ebb3da14}
   Get Get: Id {884afb94-efd9-439f-bae0-ba17499a176f}
   Set Set: Id {3a58c369-418e-4c69-93da-10a00e2004ff}
   Property MoverJerk: Id {5a9d4136-5d1c-4a75-87a5-d8c9624b6c9e}
   Get Get: Id {b43c6ed6-c2d3-4a6f-931b-a00f7c04025f}
   Set Set: Id {696042f5-0b2f-4a29-8189-8bd8a33370cb}
   Property MoverVelocity: Id {742b6ed5-8994-47d0-9514-f9da80a4d053}
   Get Get: Id {a39c28bf-5625-4f47-9c93-b9492438d570}
   Set Set: Id {d4daa692-d037-4d79-8e53-0169ed18b08c}
   Property NumberOfRotations: Id {bb4ff67d-7367-4b7a-959f-713804187620}
   Get Get: Id {5b9291ce-f4c0-4cba-bab1-5877eaf99aad}
   Set Set: Id {d5eb936f-7c12-4a48-8ac9-c0d81b0e38d0}
   Method ResetErrors: Id {3c8381a0-95d7-49ca-b1ac-a766e6689e5f}
   Method Spin: Id {c0469bb5-8daf-4d6a-9025-07ed0e9b795c}
   Method SwapPlaces: Id {2b69bc2c-8a8e-489d-9688-bbcbb0285218}
   Method Tilt: Id {42665e86-4a61-4716-bd60-3a2489faf341}
   Method VaryMoverHeight: Id {3f462c74-2326-4182-a953-36e0d5d57b05} *)
